// TIA Portal V20 export
TYPE "LER_typeAlignSyncMoveConfiguration"
// stored: Access Published
   STRUCT
      MoveDeg : LReal;
      MoveYPosition : LReal;
   END_STRUCT;
END_TYPE
